PROGRAM Q4
VAR
	// num1 := 1;
	// Missing DataType
	num1 : INT := 1;
END_VAR

END_PROGRAM

(* stored: Version 1.1.0.1, ProductVersion 3.1.4024.12
   POU Q4: Id {94a8fcd4-1478-4983-9cff-294f0b208105}, SpecialFunc None *)
